(*

## Short summary
This class provides assert statements for unsigned short integers  (``USINT``)

.. <legal notes>

legal notes
=================
| SPDX-FileCopyrightText: © 2022 ekvip automation GmbH <info@ekvip.de>
| SPDX-License-Identifier: Apache-2.0
| For details check: Apache-2.0_

.. _Apache-2.0: https://www.apache.org/licenses/LICENSE-2.0

.. </legal notes>

*)

{attribute 'reflection'}
FUNCTION_BLOCK INTERNAL UsintAssertions EXTENDS AbstractAssertion IMPLEMENTS IUsintAssertions
VAR
END_VAR
VAR CONSTANT
	LSB_MASK :USINT := 1;
END_VAR

(*

## Short summary
This abstract property returns the class name of the concrete object, 
It's for debugging purpose

.. <legal notes>

legal notes
=================
| SPDX-FileCopyrightText: © 2022 ekvip automation GmbH <info@ekvip.de>
| SPDX-License-Identifier: Apache-2.0
| For details check: Apache-2.0_

.. _Apache-2.0: https://www.apache.org/licenses/LICENSE-2.0

.. </legal notes>

*)

PROPERTY className :CNM_AbstractObject.ClassName
GET
className := 'CNM_Assertor.UsintAssertions';
END_GET
END_PROPERTY

(*

## Short summary
This assertion method checks if the current value is equal to the expected value

.. <legal notes>

legal notes
=================
| SPDX-FileCopyrightText: © 2022 ekvip automation GmbH <info@ekvip.de>
| SPDX-License-Identifier: Apache-2.0
| For details check: Apache-2.0_

.. _Apache-2.0: https://www.apache.org/licenses/LICENSE-2.0

.. </legal notes>



*)

METHOD valueIsEqualTo
VAR_INPUT
	(* current value to check *)
	currentValue	:USINT;
	(* expected value to compare *)
	expectedValue	:USINT;
	(* message if the assertion is false *)
	message			:AssertMessage;
END_VAR
IF (currentValue <> expectedValue) THEN
	THIS^.assertionWasWrong(message, THIS^.getDebugInfo('valueIsEqualTo'));
END_IF
END_METHOD

(*

## Short summary
This assertion method checks if the current value is even

.. <legal notes>

legal notes
=================
| SPDX-FileCopyrightText: © 2022 ekvip automation GmbH <info@ekvip.de>
| SPDX-License-Identifier: Apache-2.0
| For details check: Apache-2.0_

.. _Apache-2.0: https://www.apache.org/licenses/LICENSE-2.0

.. </legal notes>



*)

METHOD valueIsEven
VAR_INPUT
	(* current value to check *)
	currentValue	:USINT;
	(* message if the assertion is false *)
	message			:Tc2_System.T_MaxString;
END_VAR
IF ((currentValue AND THIS^.LSB_MASK) <> 0) THEN
	THIS^.assertionWasWrong(message, THIS^.getDebugInfo('valueIsEven'));
END_IF
END_METHOD

(*

## Short summary
This assertion method checks if the current value is greater than the less value

.. <legal notes>

legal notes
=================
| SPDX-FileCopyrightText: © 2022 ekvip automation GmbH <info@ekvip.de>
| SPDX-License-Identifier: Apache-2.0
| For details check: Apache-2.0_

.. _Apache-2.0: https://www.apache.org/licenses/LICENSE-2.0

.. </legal notes>



*)

METHOD valueIsGreaterThan
VAR_INPUT
	(* current value to check *)
	currentValue	:USINT;
	(* less than lower limit *)
	lessValue		:USINT;
	(* message if the assertion is false *)
	message			:AssertMessage;
END_VAR
IF (currentValue <= lessValue) THEN
	THIS^.assertionWasWrong(message, THIS^.getDebugInfo('valueIsGreaterThan'));
END_IF
END_METHOD

(*

## Short summary
This assertion method checks if the current value is inside a limit

**Attention:** 
	limits are included: ``valueIsInRangeOf(3, 3, 3)`` is a true assertion

.. <legal notes>

legal notes
=================
| SPDX-FileCopyrightText: © 2022 ekvip automation GmbH <info@ekvip.de>
| SPDX-License-Identifier: Apache-2.0
| For details check: Apache-2.0_

.. _Apache-2.0: https://www.apache.org/licenses/LICENSE-2.0

.. </legal notes>



*)

METHOD valueIsInRangeOf
VAR_INPUT
	(* lower limit for the current value *)
	lowerLimit		:USINT;
	(* current value to check *)
	currentValue	:USINT;
	(* upper limit for the current value *)
	upperLimit		:USINT;
	(* message if the assertion is false *)
	message			:AssertMessage;
END_VAR
IF (
	(currentValue < lowerLimit)
	OR_ELSE (currentValue > upperLimit)
) THEN
	THIS^.assertionWasWrong(message, THIS^.getDebugInfo('valueIsInRangeOf'));
END_IF
END_METHOD

(*

## Short summary
This assertion method checks if the current value is less than the greater value

.. <legal notes>

legal notes
=================
| SPDX-FileCopyrightText: © 2022 ekvip automation GmbH <info@ekvip.de>
| SPDX-License-Identifier: Apache-2.0
| For details check: Apache-2.0_

.. _Apache-2.0: https://www.apache.org/licenses/LICENSE-2.0

.. </legal notes>



*)

METHOD valueIsLessThan
VAR_INPUT
	(* current value to check *)
	currentValue	:USINT;
	(* greater than upper limit *)
	greaterValue	:USINT;
	(* message if the assertion is false *)
	message			:AssertMessage;
END_VAR
IF (currentValue >= greaterValue) THEN
	THIS^.assertionWasWrong(message, THIS^.getDebugInfo('valueIsLessThan'));
END_IF
END_METHOD

(*

## Short summary
This assertion method checks if the current value is less than or equal to the maximum value

.. <legal notes>

legal notes
=================
| SPDX-FileCopyrightText: © 2022 ekvip automation GmbH <info@ekvip.de>
| SPDX-License-Identifier: Apache-2.0
| For details check: Apache-2.0_

.. _Apache-2.0: https://www.apache.org/licenses/LICENSE-2.0

.. </legal notes>



*)

METHOD valueIsMax
VAR_INPUT
	(* current value to check *)
	currentValue	:USINT;
	(* upper limit for the current value *)
	maximumValue	:USINT;
	(* message if the assertion is false *)
	message			:AssertMessage;
END_VAR
IF (currentValue > maximumValue) THEN
	THIS^.assertionWasWrong(message, THIS^.getDebugInfo('valueIsMax'));
END_IF
END_METHOD

(*

## Short summary
This assertion method checks if the current value is greater than or equal to the minimum value

.. <legal notes>

legal notes
=================
| SPDX-FileCopyrightText: © 2022 ekvip automation GmbH <info@ekvip.de>
| SPDX-License-Identifier: Apache-2.0
| For details check: Apache-2.0_

.. _Apache-2.0: https://www.apache.org/licenses/LICENSE-2.0

.. </legal notes>



*)

METHOD valueIsMin
VAR_INPUT
	(* current value to check *)
	currentValue	:USINT;
	(* lower limit for the current value *)
	minimumValue	:USINT;
	(* message if the assertion is false *)
	message			:AssertMessage;
END_VAR
IF (currentValue < minimumValue) THEN
	THIS^.assertionWasWrong(message, THIS^.getDebugInfo('valueIsMin'));
END_IF
END_METHOD

(*

## Short summary
This assertion method checks if the current value is not equal to the unexpected value

.. <legal notes>

legal notes
=================
| SPDX-FileCopyrightText: © 2022 ekvip automation GmbH <info@ekvip.de>
| SPDX-License-Identifier: Apache-2.0
| For details check: Apache-2.0_

.. _Apache-2.0: https://www.apache.org/licenses/LICENSE-2.0

.. </legal notes>



*)

METHOD valueIsNotEqualTo
VAR_INPUT
	(* current value to check *)
	currentValue	:USINT;
	(* unexpected value to compare *)
	unexpectedValue	:USINT;
	(* message if the assertion is false *)
	message			:AssertMessage;
END_VAR
IF (currentValue = unexpectedValue) THEN
	THIS^.assertionWasWrong(message, THIS^.getDebugInfo('valueIsNotEqualTo'));
END_IF
END_METHOD

(*

## Short summary
This assertion method checks if the current value is odd

.. <legal notes>

legal notes
=================
| SPDX-FileCopyrightText: © 2022 ekvip automation GmbH <info@ekvip.de>
| SPDX-License-Identifier: Apache-2.0
| For details check: Apache-2.0_

.. _Apache-2.0: https://www.apache.org/licenses/LICENSE-2.0

.. </legal notes>



*)

METHOD valueIsOdd
VAR_INPUT
	(* current value to check *)
	currentValue	:USINT;
	(* message if the assertion is false *)
	message			:AssertMessage;
END_VAR
IF ((currentValue AND THIS^.LSB_MASK) = 0) THEN
	THIS^.assertionWasWrong(message, THIS^.getDebugInfo('valueIsOdd'));
END_IF
END_METHOD

END_FUNCTION_BLOCK

(* stored: Version 1.1.0.1, ProductVersion 3.1.4026.11
   POU UsintAssertions: Id {b16577be-b233-4f51-a2e9-1df6fe4a1e39}, SpecialFunc None
   Property className: Id {ea7e8cac-4057-4832-be4c-a31ab3330c32}
   Get Get: Id {0bc1737f-e805-4fd3-bba4-f041ef34f1bb}
   Method valueIsEqualTo: Id {02ddcb60-5b80-4e1c-83f6-09c37ac19dfb}
   Method valueIsEven: Id {83fae5be-5fcf-4950-aab6-fd10c0389426}
   Method valueIsGreaterThan: Id {4de1a634-acf2-4d16-b101-930503b59480}
   Method valueIsInRangeOf: Id {0aa3782d-66f4-434e-be73-0b511543e81c}
   Method valueIsLessThan: Id {ee123074-dd12-48f6-9afe-c750bdffdf84}
   Method valueIsMax: Id {f049b621-9deb-44e1-ac3a-2bf365d7fb7a}
   Method valueIsMin: Id {1f200bf3-ed82-420e-8f69-c4682c78de7e}
   Method valueIsNotEqualTo: Id {7a4d9285-ae10-437f-a6f1-0ef9e36879dd}
   Method valueIsOdd: Id {3c44dcfa-6807-4cd9-96d3-c94b4faf34a8} *)
